// SIMATIC S7-200 project (STEP 7-Micro/WIN), CPU 221 REL 01.10

ORGANIZATION_BLOCK 主程序:OB1
TITLE=程序注释
BEGIN
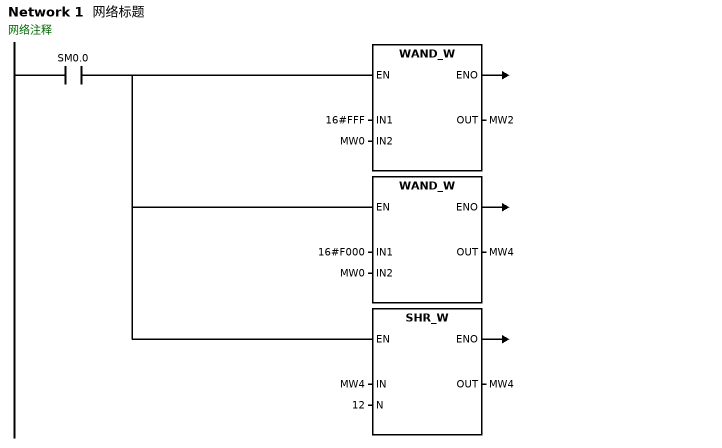
Network 1 // 网络标题
// 网络注释
// (network saved uncompiled; LAD cells follow)
// row 0: c0 -| |- SM0.0 v  c1 --  c2 --  c3 [WAND_W EN:=power@row0, IN1:=16#FFF, IN2:=MW0, ENO=>power, OUT=>MW2]  c4 ->
// row 1: c0 ^v  c3 [box]
// row 2: c0 ^v  c1 --  c2 --  c3 [WAND_W EN:=power@row2, IN1:=16#F000, IN2:=MW0, ENO=>power, OUT=>MW4]  c4 ->
// row 3: c0 ^v  c3 [box]
// row 4: c0 ^  c1 --  c2 --  c3 [SHR_W EN:=power@row4, IN:=MW4, N:=12, ENO=>power, OUT=>MW4]  c4 ->
// row 5: c3 [box]
END_ORGANIZATION_BLOCK
